% RSLogix 500 project 4P4_E_drbitboy_refactor_00.RSS, saved by version 8.30.00.16 %
PROJECT "4P4_E"    % processor: Bul.1763 MicroLogix 1100 Series B %

PROGRAM FILES
  LAD 2 "MAIN_PROG"  7 rungs
  LAD 3 "USER_FAULT"  2 rungs
  LAD 5 "INPUTCHECK"  10 rungs
  LAD 7 "DOBUSINESS"  13 rungs
  LAD 14 "OUTPUT2SIM"  3 rungs
  LAD 15 "SIMULATION"  20 rungs

DATA FILES
  O0 OUTPUT  4 elements
  I1 INPUT  6 elements
  S2 STATUS  66 elements
  B3 BINARY  32 elements
  T4 TIMER  40 elements
  C5 COUNTER  32 elements
  R6 CONTROL  16 elements
  N7 INTEGER  105 elements
  F8 FLOAT  1 elements

LADDER 2 "MAIN_PROG"
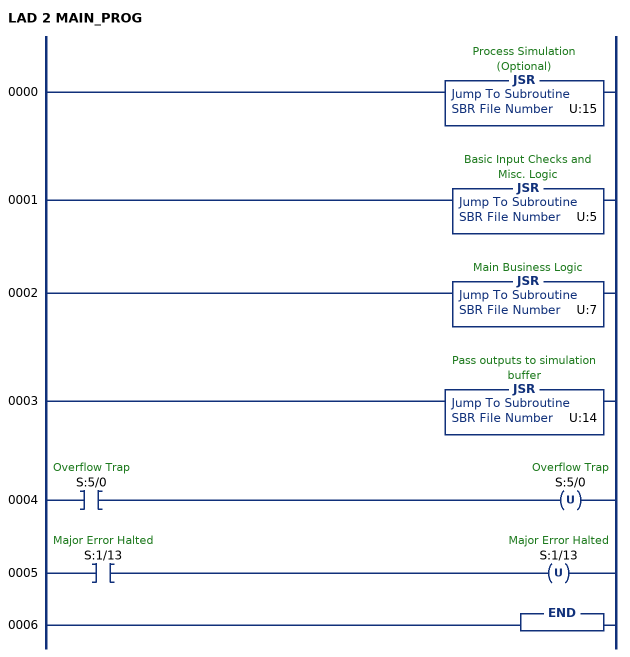
% Rung: 0 %
SOR JSR U:15 EOR
%   U:15  "Process Simulation (Optional)" %
% Rung: 1 %
SOR JSR U:5 EOR
%   U:5  "Basic Input Checks and Misc. Logic" %
% Rung: 2 %
SOR JSR U:7 EOR
%   U:7  "Main Business Logic" %
% Rung: 3 %
SOR JSR U:14 EOR
%   U:14  "Pass outputs to simulation buffer" %
% Rung: 4 %
SOR XIC S:5/0 OTU S:5/0 EOR
%   S:5/0  "Overflow Trap" %
% Rung: 5 %
SOR XIC S:1/13 OTU S:1/13 EOR
%   S:1/13  "Major Error Halted" %
% Rung: 6 %
SOR END EOR

LADDER 3 "USER_FAULT"
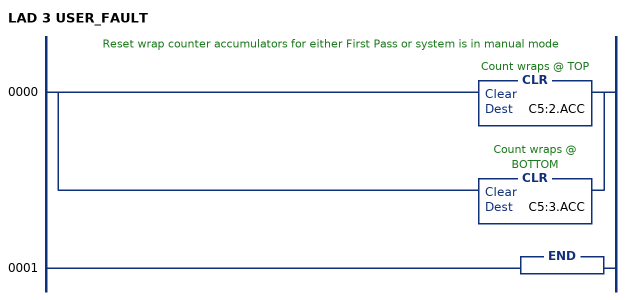
% Rung: 0 %
% Reset wrap counter accumulators for either First Pass or system is in manual mode %
SOR BST CLR C5:2.ACC NXB CLR C5:3.ACC BND EOR
%   C5:2  "Count wraps @ TOP" %
%   C5:3  "Count wraps @ BOTTOM" %
% Rung: 1 %
SOR END EOR

LADDER 5 "INPUTCHECK"
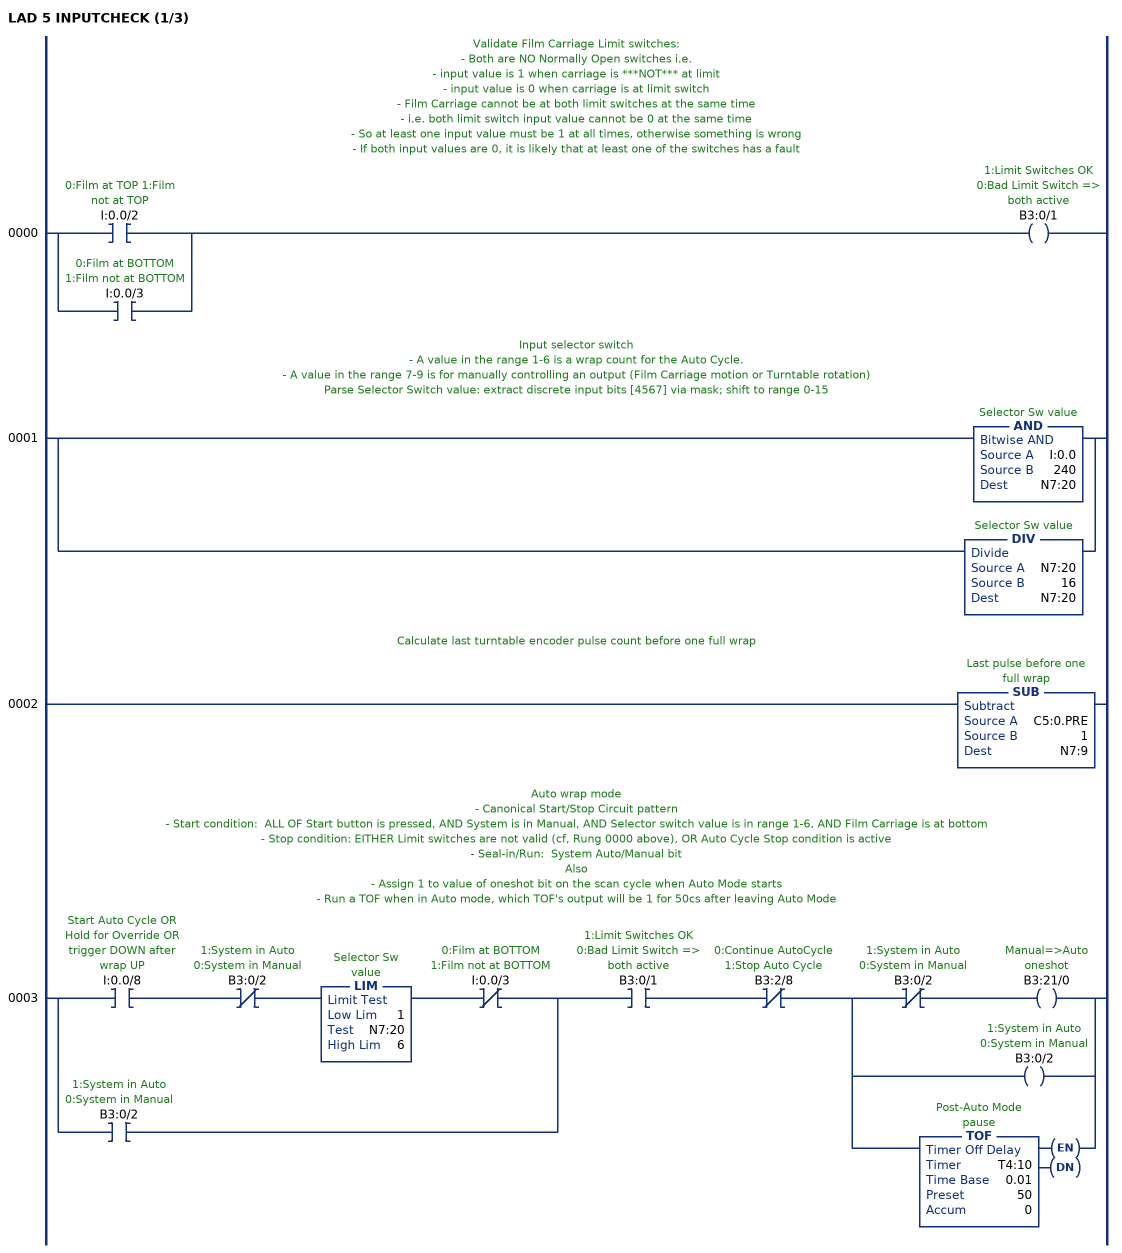
% Rung: 0 %
% Validate Film Carriage Limit switches:
% - Both are NO Normally Open switches i.e.
%   - input value is 1 when carriage is ***NOT*** at limit
%   - input value is 0 when carriage is at limit switch
% - Film Carriage cannot be at both limit switches at the same time
%   - i.e. both limit switch input value cannot be 0 at the same time
%   - So at least one input value must be 1 at all times, otherwise something is wrong
% - If both input values are 0, it is likely that at least one of the switches has a fault %
SOR BST XIC I:0.0/2 NXB XIC I:0.0/3 BND OTE B3:0/1 EOR
%   I:0.0/2  "0:Film at TOP 1:Film not at TOP" %
%   XIC I:0.0/2  "1:Film not at TOP" %
%   I:0.0/3  "0:Film at BOTTOM 1:Film not at BOTTOM" %
%   XIC I:0.0/3  "1:Film not at BOTTOM" %
%   B3:0/1  "1:Limit Switches OK 0:Bad Limit Switch => both active" %
% Rung: 1 %
% Input selector switch
% - A value in the range 1-6 is a wrap count for the Auto Cycle.
% - A value in the range 7-9 is for manually controlling an output (Film Carriage motion or Turntable rotation)
% 
% Parse Selector Switch value: extract discrete input bits [4567] via mask; shift to range 0-15 %
SOR BST AND I:0.0 240 N7:20 NXB DIV N7:20 16 N7:20 BND EOR
%   I:0.0  "INPUT Word" %
%   N7:20  "Selector Sw value" %
% Rung: 2 %
% Calculate last turntable encoder pulse count before one full wrap %
SOR SUB C5:0.PRE 1 N7:9 EOR
%   C5:0  "Count turntable pulses 112 per wrap?" %
%   N7:9  "Last pulse before one full wrap" %
% Rung: 3 %
% Auto wrap mode
% - Canonical Start/Stop Circuit pattern
%   - Start condition:  ALL OF Start button is pressed, AND System is in Manual, AND Selector switch value is in range 1-6, AND Film Carriage is at bottom
%   - Stop condition: EITHER Limit switches are not valid (cf, Rung 0000 above), OR Auto Cycle Stop condition is active
%   - Seal-in/Run:  System Auto/Manual bit
% Also
% - Assign 1 to value of oneshot bit on the scan cycle when Auto Mode starts
% - Run a TOF when in Auto mode, which TOF's output will be 1 for 50cs after leaving Auto Mode %
SOR BST XIC I:0.0/8 XIO B3:0/2 LIM 1 N7:20 6 XIO I:0.0/3 NXB XIC B3:0/2 BND XIC B3:0/1 XIO B3:2/8 BST XIO B3:0/2 OTE B3:21/0 NXB OTE B3:0/2 NXB TOF T4:10 0.01 50 0 BND EOR
%   I:0.0/8  "Start Auto Cycle OR Hold for Override OR trigger DOWN after wrap UP" %
%   B3:0/2  "1:System in Auto 0:System in Manual" %
%   XIO B3:0/2  "0:System in Manual" %
%   N7:20  "Selector Sw value" %
%   I:0.0/3  "0:Film at BOTTOM 1:Film not at BOTTOM" %
%   XIO I:0.0/3  "0:Film at BOTTOM" %
%   XIC B3:0/2  "1:System in Auto" %
%   B3:0/1  "1:Limit Switches OK 0:Bad Limit Switch => both active" %
%   XIC B3:0/1  "1:Limit Switches OK" %
%   B3:2/8  "0:Continue AutoCycle 1:Stop Auto Cycle" %
%   B3:21/0  "Manual=>Auto oneshot" %
%   T4:10  "Post-Auto Mode pause" %

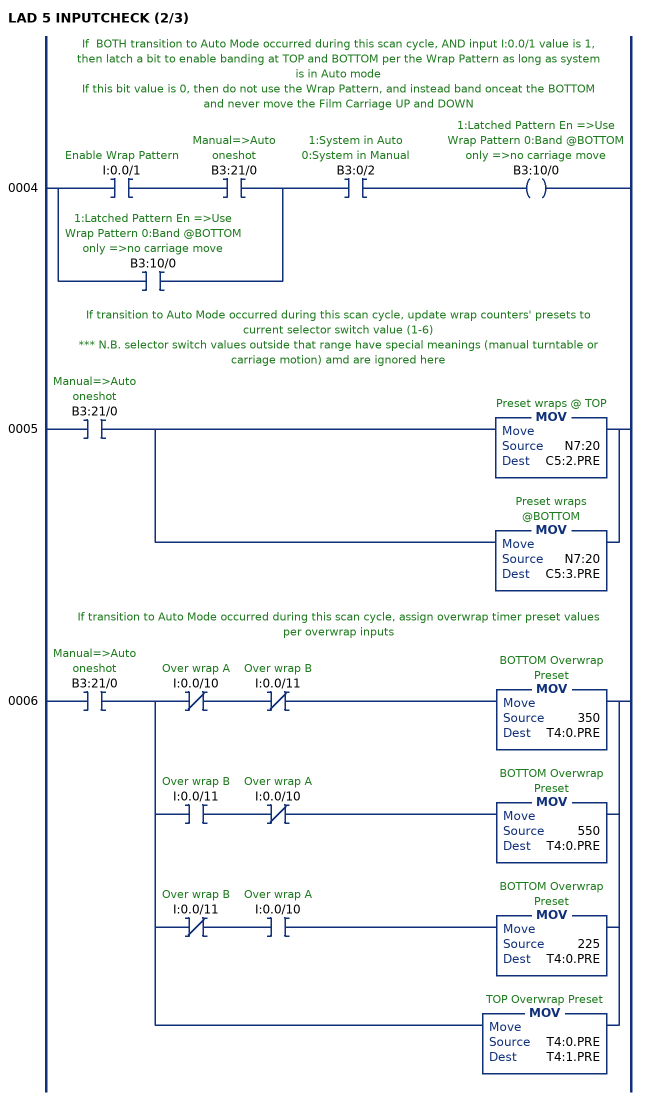
% Rung: 4 %
% If  BOTH transition to Auto Mode occurred during this scan cycle, AND input I:0.0/1 value is 1, then latch a bit to enable banding at TOP and BOTTOM per the Wrap Pattern as long as system is in Auto mode
% If this bit value is 0, then do not use the Wrap Pattern, and instead band onceat the BOTTOM and never move the Film Carriage UP and DOWN %
SOR BST XIC I:0.0/1 XIC B3:21/0 NXB XIC B3:10/0 BND XIC B3:0/2 OTE B3:10/0 EOR
%   I:0.0/1  "Enable Wrap Pattern" %
%   B3:21/0  "Manual=>Auto oneshot" %
%   B3:10/0  "1:Latched Pattern En =>Use Wrap Pattern 0:Band @BOTTOM only =>no carriage move" %
%   XIC B3:10/0  "1:Latched Pattern En =>Use Wrap Pattern =>In Auto Mode" %
%   B3:0/2  "1:System in Auto 0:System in Manual" %
%   XIC B3:0/2  "1:System in Auto" %
% Rung: 5 %
% If transition to Auto Mode occurred during this scan cycle, update wrap counters' presets to current selector switch value (1-6)
% *** N.B. selector switch values outside that range have special meanings (manual turntable or carriage motion) amd are ignored here %
SOR XIC B3:21/0 BST MOV N7:20 C5:2.PRE NXB MOV N7:20 C5:3.PRE BND EOR
%   B3:21/0  "Manual=>Auto oneshot" %
%   N7:20  "Selector Sw value" %
%   C5:2.PRE  "Preset wraps @ TOP" %
%   C5:3.PRE  "Preset wraps @BOTTOM" %
% Rung: 6 %
% If transition to Auto Mode occurred during this scan cycle, assign overwrap timer preset values per overwrap inputs %
SOR XIC B3:21/0 BST XIO I:0.0/10 XIO I:0.0/11 MOV 350 T4:0.PRE NXB XIC I:0.0/11 XIO I:0.0/10 MOV 550 T4:0.PRE NXB XIO I:0.0/11 XIC I:0.0/10 MOV 225 T4:0.PRE NXB MOV T4:0.PRE T4:1.PRE BND EOR
%   B3:21/0  "Manual=>Auto oneshot" %
%   I:0.0/10  "Over wrap A" %
%   I:0.0/11  "Over wrap B" %
%   T4:0.PRE  "BOTTOM Overwrap Preset" %
%   T4:1.PRE  "TOP Overwrap Preset" %

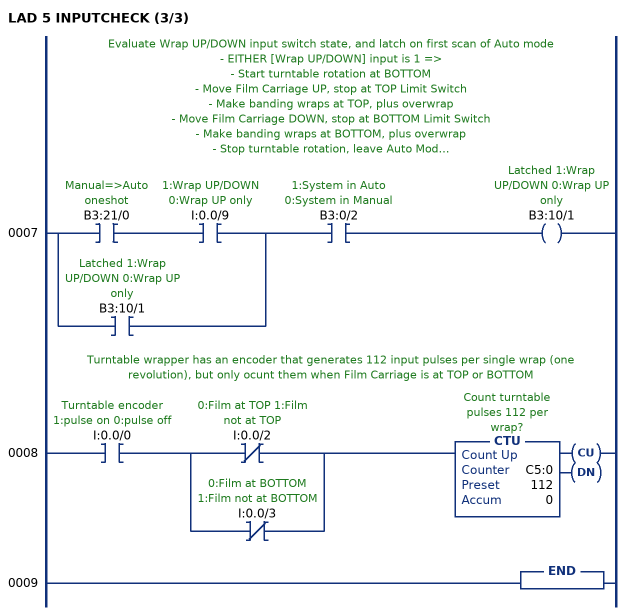
% Rung: 7 %
% Evaluate Wrap UP/DOWN input switch state, and latch on first scan of Auto mode
% - EITHER [Wrap UP/DOWN] input is 1 =>
%   - Start turntable rotation at BOTTOM
%   - Move Film Carriage UP, stop at TOP Limit Switch
%   - Make banding wraps at TOP, plus overwrap
%   - Move Film Carriage DOWN, stop at BOTTOM Limit Switch
%   - Make banding wraps at BOTTOM, plus overwrap
%   - Stop turntable rotation, leave Auto Mode
% - OR [Wrap UP/DOWN] input is 0 (Wrap UP only) =>
%   - Start turntable rotation at BOTTOM
%   - Make banding wraps at BOTTOM, plus overwrap
%   - Move File Carriage UP, stop at TOP Limit Switch
%   - Make banding wraps at TOP, plus overwrap
%   - Stop Turntable rotation
%   - Flash light, wait for operator to (cut film and then) press Start
%   - Move Film Carriage DOWN, stop at BOTTOM Limit Switch
%   - Leave Auto Mode %
SOR BST XIC B3:21/0 XIC I:0.0/9 NXB XIC B3:10/1 BND XIC B3:0/2 OTE B3:10/1 EOR
%   B3:21/0  "Manual=>Auto oneshot" %
%   I:0.0/9  "1:Wrap UP/DOWN 0:Wrap UP only" %
%   B3:10/1  "Latched 1:Wrap UP/DOWN 0:Wrap UP only" %
%   XIC B3:10/1  "Latched 1:Wrap UP/DOWN" %
%   B3:0/2  "1:System in Auto 0:System in Manual" %
%   XIC B3:0/2  "1:System in Auto" %
% Rung: 8 %
% Turntable wrapper has an encoder that generates 112 input pulses per single wrap (one revolution), but only ocunt them when Film Carriage is at TOP or BOTTOM %
SOR XIC I:0.0/0 BST XIO I:0.0/2 NXB XIO I:0.0/3 BND CTU C5:0 112 0 EOR
%   I:0.0/0  "Turntable encoder 1:pulse on 0:pulse off" %
%   XIC I:0.0/0  "1:Turntable encoder pulse on" %
%   I:0.0/2  "0:Film at TOP 1:Film not at TOP" %
%   XIO I:0.0/2  "0:Film at TOP" %
%   I:0.0/3  "0:Film at BOTTOM 1:Film not at BOTTOM" %
%   XIO I:0.0/3  "0:Film at BOTTOM" %
%   C5:0  "Count turntable pulses 112 per wrap?" %
% Rung: 9 %
SOR END EOR

LADDER 7 "DOBUSINESS"
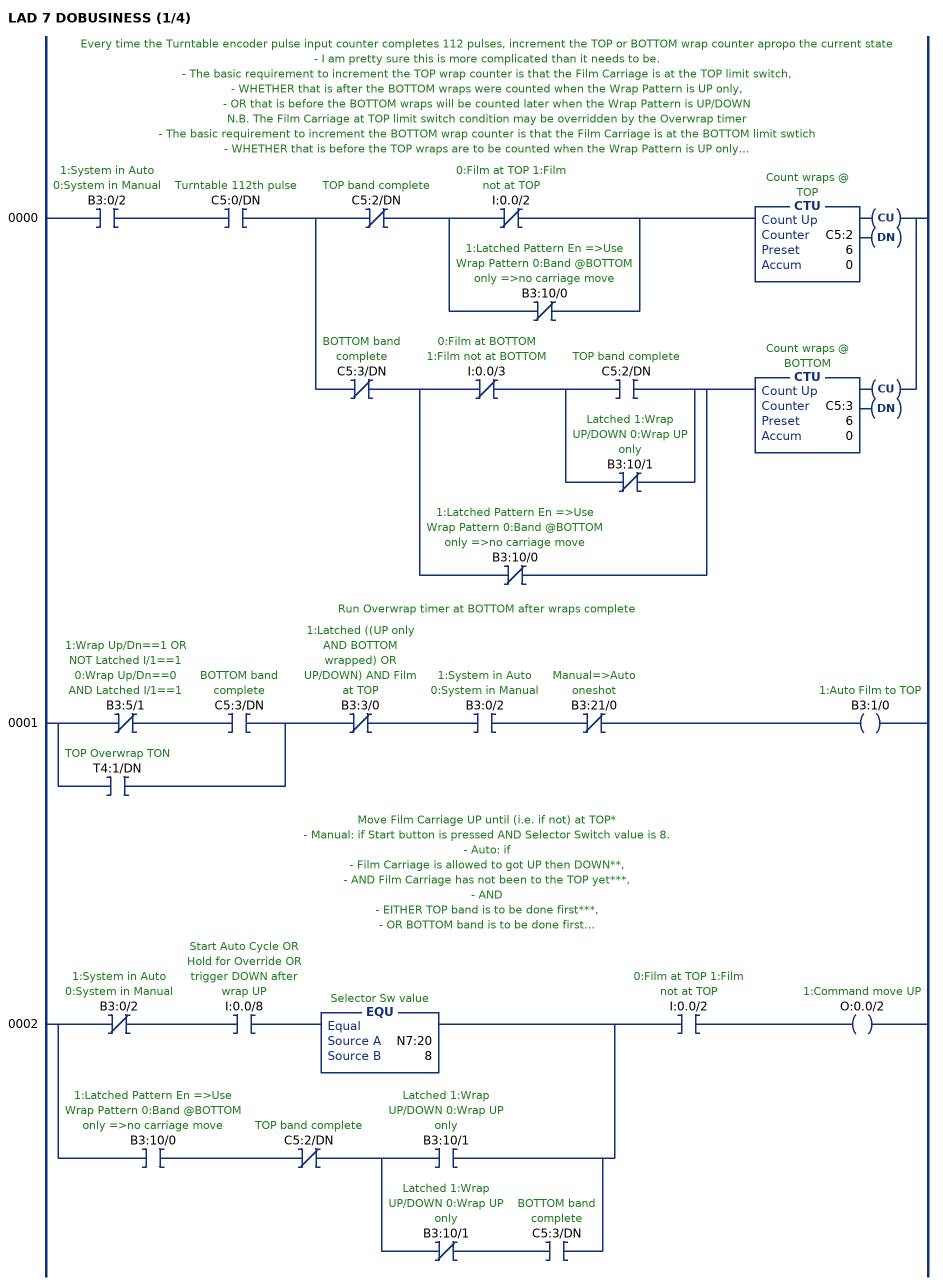
% Rung: 0 %
% Every time the Turntable encoder pulse input counter completes 112 pulses, increment the TOP or BOTTOM wrap counter apropo the current state
% - I am pretty sure this is more complicated than it needs to be.
% 
% - The basic requirement to increment the TOP wrap counter is that the Film Carriage is at the TOP limit switch,
%   - WHETHER that is after the BOTTOM wraps were counted when the Wrap Pattern is UP only,
%   - OR that is before the BOTTOM wraps will be counted later when the Wrap Pattern is UP/DOWN
% N.B. The Film Carriage at TOP limit switch condition may be overridden by the Overwrap timer
% 
% - The basic requirement to increment the BOTTOM wrap counter is that the Film Carriage is at the BOTTOM limit swtich
%   - WHETHER that is before the TOP wraps are to be counted when the Wrap Pattern is UP only,
%   - OR that is after the TOP wraps were counted when the Wrap Pattern is UP/DOWN
% N.B. the TOP wraps completed check for Wrap Pattern UP/DOWN may be overriden by the T4:6 timer done bit when inpu I:0.0/1 value is 0 %
SOR XIC B3:0/2 XIC C5:0/DN BST XIO C5:2/DN BST XIO I:0.0/2 NXB XIO B3:10/0 BND CTU C5:2 6 0 NXB XIO C5:3/DN BST XIO I:0.0/3 BST XIC C5:2/DN NXB XIO B3:10/1 BND NXB XIO B3:10/0 BND CTU C5:3 6 0 BND EOR
%   B3:0/2  "1:System in Auto 0:System in Manual" %
%   XIC B3:0/2  "1:System in Auto" %
%   C5:0/DN  "Turntable 112th pulse" %
%   C5:2/DN  "TOP band complete" %
%   XIO C5:2/DN  "TOP band incomplete" %
%   I:0.0/2  "0:Film at TOP 1:Film not at TOP" %
%   XIO I:0.0/2  "0:Film at TOP" %
%   B3:10/0  "1:Latched Pattern En =>Use Wrap Pattern 0:Band @BOTTOM only =>no carriage move" %
%   XIO B3:10/0  "0:Band @BOTTOM only =>no carriage move" %
%   C5:2  "Count wraps @ TOP" %
%   C5:3/DN  "BOTTOM band complete" %
%   XIO C5:3/DN  "BOTTOM band incomplete" %
%   I:0.0/3  "0:Film at BOTTOM 1:Film not at BOTTOM" %
%   XIO I:0.0/3  "0:Film at BOTTOM" %
%   B3:10/1  "Latched 1:Wrap UP/DOWN 0:Wrap UP only" %
%   XIO B3:10/1  "Latched 0:Wrap UP only" %
%   C5:3  "Count wraps @ BOTTOM" %
% Rung: 1 %
% Run Overwrap timer at BOTTOM after wraps complete %
SOR BST XIO B3:5/1 XIC C5:3/DN NXB XIC T4:1/DN BND XIO B3:3/0 XIC B3:0/2 XIO B3:21/0 OTE B3:1/0 EOR
%   B3:5/1  "1:Wrap Up/Dn==1 OR NOT Latched I/1==1 0:Wrap Up/Dn==0 AND Latched I/1==1" %
%   XIO B3:5/1  "0:Wrap UP only AND Latched I/1==1" %
%   C5:3/DN  "BOTTOM band complete" %
%   T4:1  "TOP Overwrap TON" %
%   B3:3/0  "1:Latched ((UP only AND BOTTOM wrapped) OR UP/DOWN) AND Film at TOP" %
%   B3:0/2  "1:System in Auto 0:System in Manual" %
%   XIC B3:0/2  "1:System in Auto" %
%   B3:21/0  "Manual=>Auto oneshot" %
%   XIO B3:21/0  "0:Start btn released in Auto mode" %
%   B3:1/0  "1:Auto Film to TOP" %
% Rung: 2 %
% Move Film Carriage UP until (i.e. if not) at TOP*
% - Manual: if Start button is pressed AND Selector Switch value is 8.
% - Auto: if
%   - Film Carriage is allowed to got UP then DOWN**,
%   - AND Film Carriage has not been to the TOP yet***,
%   - AND
%     - EITHER TOP band is to be done first***,
%     - OR BOTTOM band is to be done first.
% 
% * Don't need to check if Limit Switches are OK because [Film not at TOP] ensures they are
% ** [Latched Wrap Pattern Enabled] is only 1 if already in Auto Mode
% *** [TOP band incomplete] will be 1when to stop Film Carriage moving up when it is at BOTTOM the second time for [Wrap UP/DOWN]. %
SOR BST XIO B3:0/2 XIC I:0.0/8 EQU N7:20 8 NXB XIC B3:10/0 XIO C5:2/DN BST XIC B3:10/1 NXB XIO B3:10/1 XIC C5:3/DN BND BND XIC I:0.0/2 OTE O:0.0/2 EOR
%   B3:0/2  "1:System in Auto 0:System in Manual" %
%   XIO B3:0/2  "0:System in Manual" %
%   I:0.0/8  "Start Auto Cycle OR Hold for Override OR trigger DOWN after wrap UP" %
%   N7:20  "Selector Sw value" %
%   B3:10/0  "1:Latched Pattern En =>Use Wrap Pattern 0:Band @BOTTOM only =>no carriage move" %
%   XIC B3:10/0  "1:Latched Pattern En =>Use Wrap Pattern =>In Auto Mode" %
%   C5:2/DN  "TOP band complete" %
%   XIO C5:2/DN  "TOP band incomplete" %
%   B3:10/1  "Latched 1:Wrap UP/DOWN 0:Wrap UP only" %
%   XIC B3:10/1  "Latched 1:Wrap UP/DOWN" %
%   XIO B3:10/1  "Latched 0:Wrap UP only" %
%   C5:3/DN  "BOTTOM band complete" %
%   I:0.0/2  "0:Film at TOP 1:Film not at TOP" %
%   XIC I:0.0/2  "1:Film not at TOP" %
%   O:0.0/2  "1:Command move UP" %

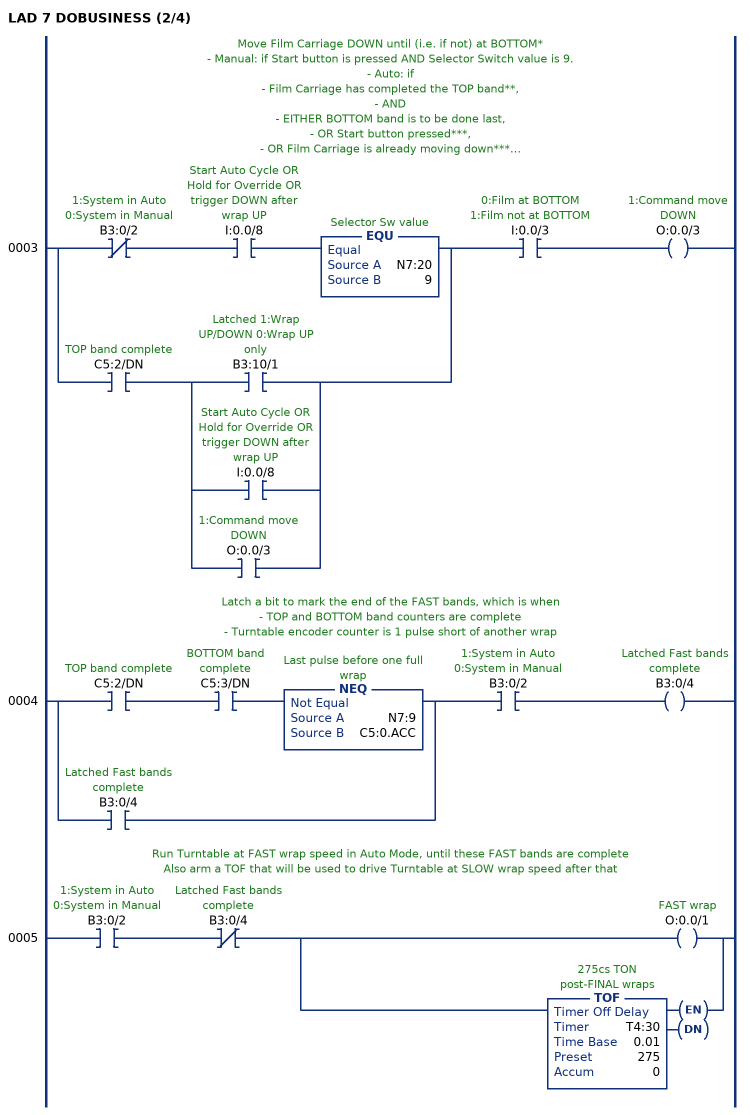
% Rung: 3 %
% Move Film Carriage DOWN until (i.e. if not) at BOTTOM*
% - Manual: if Start button is pressed AND Selector Switch value is 9.
% - Auto: if
%   - Film Carriage has completed the TOP band**,
%   - AND
%     - EITHER BOTTOM band is to be done last,
%     - OR Start button pressed***,
%     - OR Film Carriage is already moving down***.
% 
% * Don't need to check if Limit Switches are OK because [Film not at BOTTOM] ensures they are
% ** Film Carriage would not be away from BOTTOM unless [Wrap Pattern Enabled]
%   - Also TOP band can only be complete if system is in Auto Mode, because TOP band count is cleared to 0 in Manual
% *** Those last two will be the case when Wrap Pattern is Wrap UP only %
SOR BST XIO B3:0/2 XIC I:0.0/8 EQU N7:20 9 NXB XIC C5:2/DN BST XIC B3:10/1 NXB XIC I:0.0/8 NXB XIC O:0.0/3 BND BND XIC I:0.0/3 OTE O:0.0/3 EOR
%   B3:0/2  "1:System in Auto 0:System in Manual" %
%   XIO B3:0/2  "0:System in Manual" %
%   I:0.0/8  "Start Auto Cycle OR Hold for Override OR trigger DOWN after wrap UP" %
%   N7:20  "Selector Sw value" %
%   C5:2/DN  "TOP band complete" %
%   B3:10/1  "Latched 1:Wrap UP/DOWN 0:Wrap UP only" %
%   XIC B3:10/1  "Latched 1:Wrap UP/DOWN" %
%   O:0.0/3  "1:Command move DOWN" %
%   I:0.0/3  "0:Film at BOTTOM 1:Film not at BOTTOM" %
%   XIC I:0.0/3  "1:Film not at BOTTOM" %
% Rung: 4 %
% Latch a bit to mark the end of the FAST bands, which is when
% - TOP and BOTTOM band counters are complete
% - Turntable encoder counter is 1 pulse short of another wrap %
SOR BST XIC C5:2/DN XIC C5:3/DN NEQ N7:9 C5:0.ACC NXB XIC B3:0/4 BND XIC B3:0/2 OTE B3:0/4 EOR
%   C5:2/DN  "TOP band complete" %
%   C5:3/DN  "BOTTOM band complete" %
%   N7:9  "Last pulse before one full wrap" %
%   C5:0.ACC  "Turntable pulse count" %
%   B3:0/4  "Latched Fast bands complete" %
%   XIC B3:0/4  "1:Fast bands complete" %
%   B3:0/2  "1:System in Auto 0:System in Manual" %
%   XIC B3:0/2  "1:System in Auto" %
% Rung: 5 %
% Run Turntable at FAST wrap speed in Auto Mode, until these FAST bands are complete
% Also arm a TOF that will be used to drive Turntable at SLOW wrap speed after that %
SOR XIC B3:0/2 XIO B3:0/4 BST OTE O:0.0/1 NXB TOF T4:30 0.01 275 0 BND EOR
%   B3:0/2  "1:System in Auto 0:System in Manual" %
%   XIC B3:0/2  "1:System in Auto" %
%   B3:0/4  "Latched Fast bands complete" %
%   XIO B3:0/4  "0:Fast bands incomplete" %
%   O:0.0/1  "FAST wrap" %
%   T4:30  "275cs TON post-FINAL wraps" %

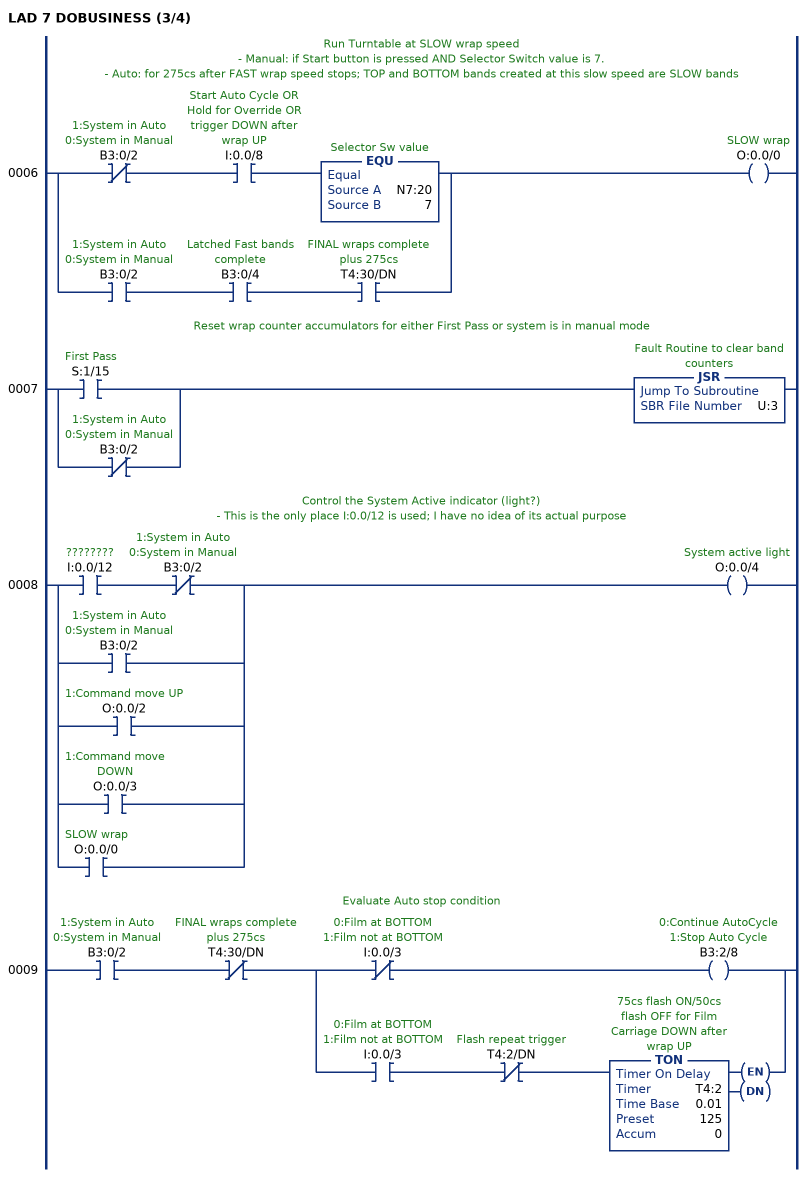
% Rung: 6 %
% Run Turntable at SLOW wrap speed
% - Manual: if Start button is pressed AND Selector Switch value is 7.
% - Auto: for 275cs after FAST wrap speed stops; TOP and BOTTOM bands created at this slow speed are SLOW bands %
SOR BST XIO B3:0/2 XIC I:0.0/8 EQU N7:20 7 NXB XIC B3:0/2 XIC B3:0/4 XIC T4:30/DN BND OTE O:0.0/0 EOR
%   B3:0/2  "1:System in Auto 0:System in Manual" %
%   XIO B3:0/2  "0:System in Manual" %
%   I:0.0/8  "Start Auto Cycle OR Hold for Override OR trigger DOWN after wrap UP" %
%   N7:20  "Selector Sw value" %
%   XIC B3:0/2  "1:System in Auto" %
%   B3:0/4  "Latched Fast bands complete" %
%   XIC B3:0/4  "1:Fast bands complete" %
%   T4:30/DN  "FINAL wraps complete plus 275cs" %
%   O:0.0/0  "SLOW wrap" %
% Rung: 7 %
% Reset wrap counter accumulators for either First Pass or system is in manual mode %
SOR BST XIC S:1/15 NXB XIO B3:0/2 BND JSR U:3 EOR
%   S:1/15  "First Pass" %
%   B3:0/2  "1:System in Auto 0:System in Manual" %
%   XIO B3:0/2  "0:System in Manual" %
%   U:3  "Fault Routine to clear band counters" %
% Rung: 8 %
% Control the System Active indicator (light?)
% - This is the only place I:0.0/12 is used; I have no idea of its actual purpose %
SOR BST XIC I:0.0/12 XIO B3:0/2 NXB XIC B3:0/2 NXB XIC O:0.0/2 NXB XIC O:0.0/3 NXB XIC O:0.0/0 BND OTE O:0.0/4 EOR
%   I:0.0/12  "????????" %
%   B3:0/2  "1:System in Auto 0:System in Manual" %
%   XIO B3:0/2  "0:System in Manual" %
%   XIC B3:0/2  "1:System in Auto" %
%   O:0.0/2  "1:Command move UP" %
%   O:0.0/3  "1:Command move DOWN" %
%   O:0.0/0  "SLOW wrap" %
%   O:0.0/4  "System active light" %
% Rung: 9 %
% Evaluate Auto stop condition %
SOR XIC B3:0/2 XIO T4:30/DN BST XIO I:0.0/3 OTE B3:2/8 NXB XIC I:0.0/3 XIO T4:2/DN TON T4:2 0.01 125 0 BND EOR
%   B3:0/2  "1:System in Auto 0:System in Manual" %
%   XIC B3:0/2  "1:System in Auto" %
%   T4:30/DN  "FINAL wraps complete plus 275cs" %
%   I:0.0/3  "0:Film at BOTTOM 1:Film not at BOTTOM" %
%   XIO I:0.0/3  "0:Film at BOTTOM" %
%   B3:2/8  "0:Continue AutoCycle 1:Stop Auto Cycle" %
%   XIC I:0.0/3  "1:Film not at BOTTOM" %
%   T4:2/DN  "Flash repeat trigger" %
%   T4:2  "75cs flash ON/50cs flash OFF for Film Carriage DOWN after wrap UP" %

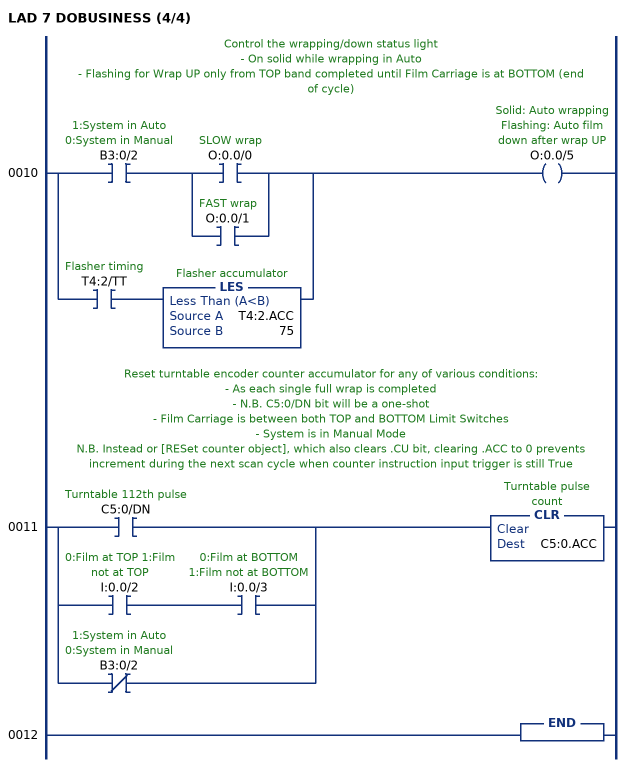
% Rung: 10 %
% Control the wrapping/down status light
% - On solid while wrapping in Auto
% - Flashing for Wrap UP only from TOP band completed until Film Carriage is at BOTTOM (end of cycle) %
SOR BST XIC B3:0/2 BST XIC O:0.0/0 NXB XIC O:0.0/1 BND NXB XIC T4:2/TT LES T4:2.ACC 75 BND OTE O:0.0/5 EOR
%   B3:0/2  "1:System in Auto 0:System in Manual" %
%   XIC B3:0/2  "1:System in Auto" %
%   O:0.0/0  "SLOW wrap" %
%   O:0.0/1  "FAST wrap" %
%   T4:2/TT  "Flasher timing" %
%   T4:2.ACC  "Flasher accumulator" %
%   O:0.0/5  "Solid: Auto wrapping Flashing: Auto film down after wrap UP" %
% Rung: 11 %
% Reset turntable encoder counter accumulator for any of various conditions:
% - As each single full wrap is completed
%   - N.B. C5:0/DN bit will be a one-shot
% - Film Carriage is between both TOP and BOTTOM Limit Switches
% - System is in Manual Mode
% N.B. Instead or [RESet counter object], which also clears .CU bit, clearing .ACC to 0 prevents
%          increment during the next scan cycle when counter instruction input trigger is still True %
SOR BST XIC C5:0/DN NXB XIC I:0.0/2 XIC I:0.0/3 NXB XIO B3:0/2 BND CLR C5:0.ACC EOR
%   C5:0/DN  "Turntable 112th pulse" %
%   I:0.0/2  "0:Film at TOP 1:Film not at TOP" %
%   XIC I:0.0/2  "1:Film not at TOP" %
%   I:0.0/3  "0:Film at BOTTOM 1:Film not at BOTTOM" %
%   XIC I:0.0/3  "1:Film not at BOTTOM" %
%   B3:0/2  "1:System in Auto 0:System in Manual" %
%   XIO B3:0/2  "0:System in Manual" %
%   C5:0.ACC  "Turntable pulse count" %
% Rung: 12 %
SOR END EOR

LADDER 14 "OUTPUT2SIM"
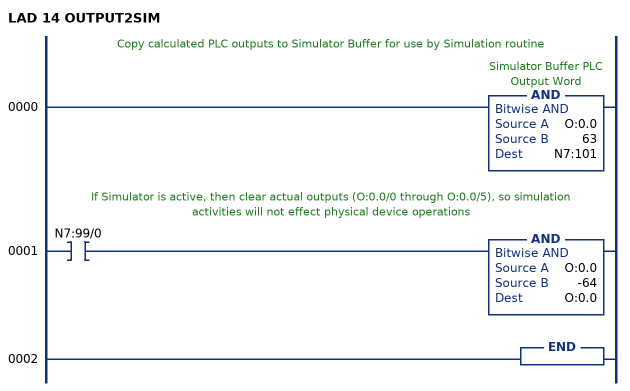
% Rung: 0 %
% Copy calculated PLC outputs to Simulator Buffer for use by Simulation routine %
SOR AND O:0.0 63 N7:101 EOR
%   N7:101  "Simulator Buffer PLC Output Word" %
% Rung: 1 %
% If Simulator is active, then clear actual outputs (O:0.0/0 through O:0.0/5), so simulation activities will not effect physical device operations %
SOR XIC N7:99/0 AND O:0.0 -64 O:0.0 EOR
% Rung: 2 %
SOR END EOR

LADDER 15 "SIMULATION"
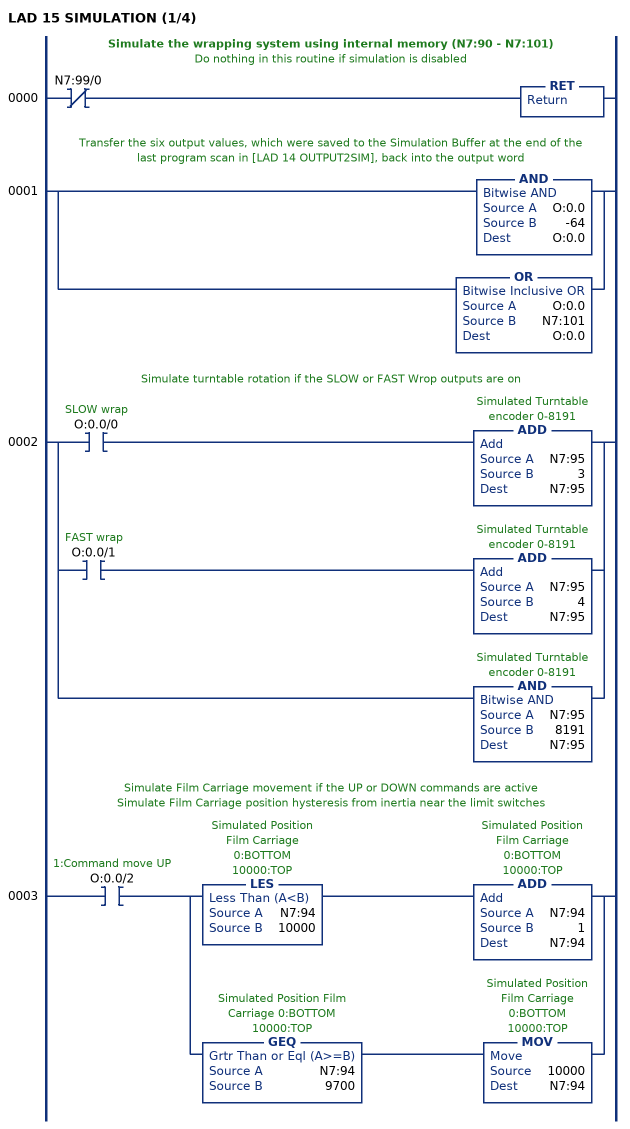
% Rung: 0 %
% TITLE: Simulate the wrapping system using internal memory (N7:90 - N7:101) %
% Do nothing in this routine if simulation is disabled %
SOR XIO N7:99/0 RET EOR
% Rung: 1 %
% Transfer the six output values, which were saved to the Simulation Buffer at the end of the last program scan in [LAD 14 OUTPUT2SIM], back into the output word %
SOR BST AND O:0.0 -64 O:0.0 NXB OR O:0.0 N7:101 O:0.0 BND EOR
%   N7:101  "Simulator Buffer PLC Output Word" %
% Rung: 2 %
% Simulate turntable rotation if the SLOW or FAST Wrop outputs are on %
SOR BST XIC O:0.0/0 ADD N7:95 3 N7:95 NXB XIC O:0.0/1 ADD N7:95 4 N7:95 NXB AND N7:95 8191 N7:95 BND EOR
%   O:0.0/0  "SLOW wrap" %
%   N7:95  "Simulated Turntable encoder 0-8191" %
%   O:0.0/1  "FAST wrap" %
% Rung: 3 %
% Simulate Film Carriage movement if the UP or DOWN commands are active
% Simulate Film Carriage position hysteresis from inertia near the limit switches %
SOR XIC O:0.0/2 BST LES N7:94 10000 ADD N7:94 1 N7:94 NXB GEQ N7:94 9700 MOV 10000 N7:94 BND EOR
%   O:0.0/2  "1:Command move UP" %
%   N7:94  "Simulated Position Film Carriage 0:BOTTOM 10000:TOP" %

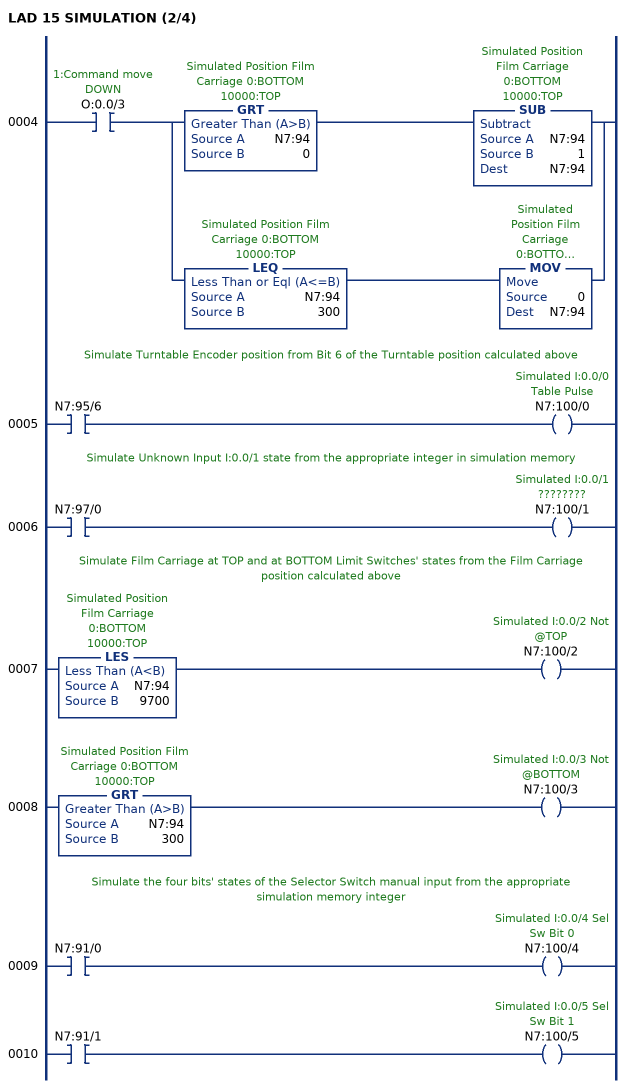
% Rung: 4 %
SOR XIC O:0.0/3 BST GRT N7:94 0 SUB N7:94 1 N7:94 NXB LEQ N7:94 300 MOV 0 N7:94 BND EOR
%   O:0.0/3  "1:Command move DOWN" %
%   N7:94  "Simulated Position Film Carriage 0:BOTTOM 10000:TOP" %
% Rung: 5 %
% Simulate Turntable Encoder position from Bit 6 of the Turntable position calculated above %
SOR XIC N7:95/6 OTE N7:100/0 EOR
%   N7:100/0  "Simulated I:0.0/0 Table Pulse" %
% Rung: 6 %
% Simulate Unknown Input I:0.0/1 state from the appropriate integer in simulation memory %
SOR XIC N7:97/0 OTE N7:100/1 EOR
%   N7:100/1  "Simulated I:0.0/1 ????????" %
% Rung: 7 %
% Simulate Film Carriage at TOP and at BOTTOM Limit Switches' states from the Film Carriage position calculated above %
SOR LES N7:94 9700 OTE N7:100/2 EOR
%   N7:94  "Simulated Position Film Carriage 0:BOTTOM 10000:TOP" %
%   N7:100/2  "Simulated I:0.0/2 Not @TOP" %
% Rung: 8 %
SOR GRT N7:94 300 OTE N7:100/3 EOR
%   N7:94  "Simulated Position Film Carriage 0:BOTTOM 10000:TOP" %
%   N7:100/3  "Simulated I:0.0/3 Not @BOTTOM" %
% Rung: 9 %
% Simulate the four bits' states of the Selector Switch manual input from the appropriate simulation memory integer %
SOR XIC N7:91/0 OTE N7:100/4 EOR
%   N7:100/4  "Simulated I:0.0/4 Sel Sw Bit 0" %
% Rung: 10 %
SOR XIC N7:91/1 OTE N7:100/5 EOR
%   N7:100/5  "Simulated I:0.0/5 Sel Sw Bit 1" %

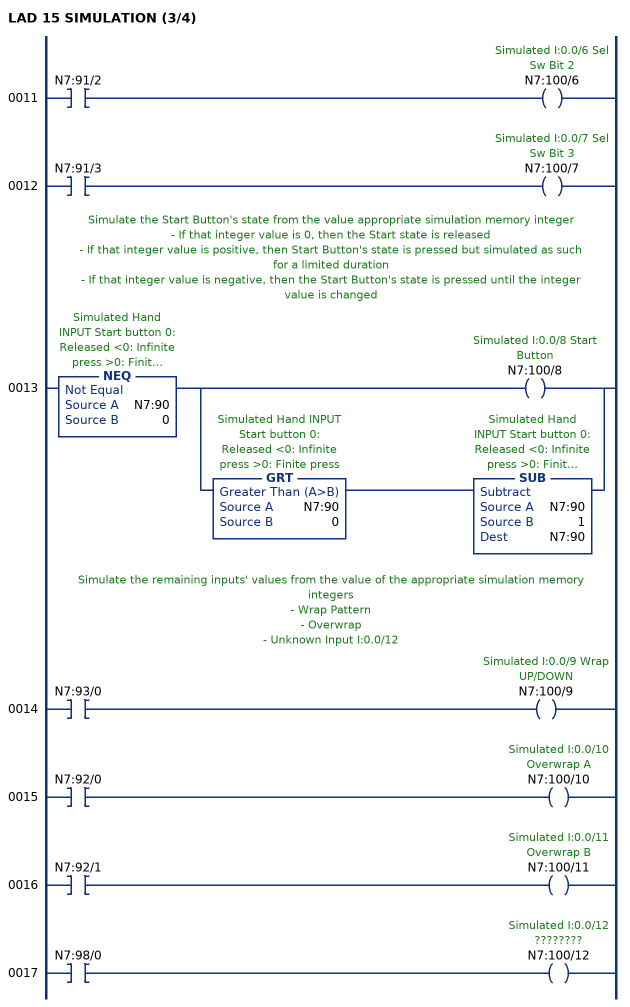
% Rung: 11 %
SOR XIC N7:91/2 OTE N7:100/6 EOR
%   N7:100/6  "Simulated I:0.0/6 Sel Sw Bit 2" %
% Rung: 12 %
SOR XIC N7:91/3 OTE N7:100/7 EOR
%   N7:100/7  "Simulated I:0.0/7 Sel Sw Bit 3" %
% Rung: 13 %
% Simulate the Start Button's state from the value appropriate simulation memory integer
% - If that integer value is 0, then the Start state is released
% - If that integer value is positive, then Start Button's state is pressed but simulated as such for a limited duration
% - If that integer value is negative, then the Start Button's state is pressed until the integer value is changed %
SOR NEQ N7:90 0 BST OTE N7:100/8 NXB GRT N7:90 0 SUB N7:90 1 N7:90 BND EOR
%   N7:90  "Simulated Hand INPUT Start button 0: Released <0: Infinite press >0: Finite press" %
%   N7:100/8  "Simulated I:0.0/8 Start Button" %
% Rung: 14 %
% Simulate the remaining inputs' values from the value of the appropriate simulation memory integers
% - Wrap Pattern
% - Overwrap
% - Unknown Input I:0.0/12 %
SOR XIC N7:93/0 OTE N7:100/9 EOR
%   N7:100/9  "Simulated I:0.0/9 Wrap UP/DOWN" %
% Rung: 15 %
SOR XIC N7:92/0 OTE N7:100/10 EOR
%   N7:100/10  "Simulated I:0.0/10 Overwrap A" %
% Rung: 16 %
SOR XIC N7:92/1 OTE N7:100/11 EOR
%   N7:100/11  "Simulated I:0.0/11 Overwrap B" %
% Rung: 17 %
SOR XIC N7:98/0 OTE N7:100/12 EOR
%   N7:100/12  "Simulated I:0.0/12 ????????" %

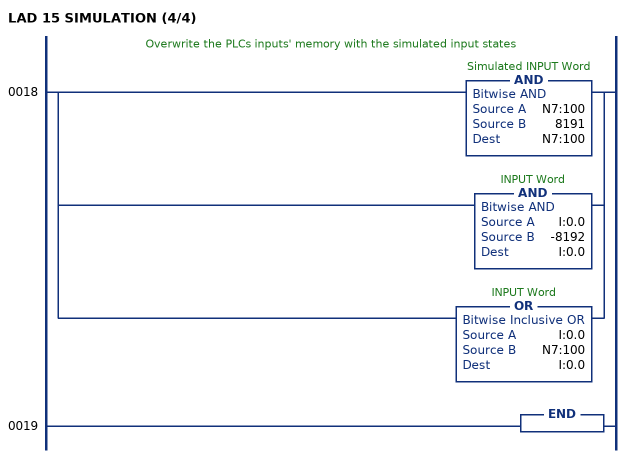
% Rung: 18 %
% Overwrite the PLCs inputs' memory with the simulated input states %
SOR BST AND N7:100 8191 N7:100 NXB AND I:0.0 -8192 I:0.0 NXB OR I:0.0 N7:100 I:0.0 BND EOR
%   N7:100  "Simulated INPUT Word" %
%   I:0.0  "INPUT Word" %
% Rung: 19 %
SOR END EOR

OTHER DOCUMENTED ADDRESSES
  B3:0/0  "1:Trigger pulse count reset"
  B3:0/3  "1:Latched FINAL wraps done + 375cs + 111 pulses 0:Continue wrapping"
  B3:0/12  "2:Latch move film DOWN after wrap UP"
  B3:1/1  "1:Wraps incomplete AND System in Auto +50cs 0:Wraps complete OR Sys in Manual"
  B3:1/8  "Film carriage DOWN trigger"
  B3:2/6  "1:Latched FINAL wraps done plus 275cs AND wrapping 0:Wraps incomplete OR NOT wrapping"
  B3:3/1  "1:Latched TOP wrapped AND film at BOTTOM"
  B3:4/0  "First-pass one-shot"
  B3:5/0  "1:Start button triggers Auto; Count switch=1-6 0:Start button other Count switch=7-9"
  B3:8/2  "Raise Film Carriage (UP override) 1: Count switch at 8 and Start pressed"
  B3:8/3  "Lower Film Carriage (DOWN override) 1: Count switch at 9 and Start pressed"
  B3:8/9  "Rotate turntable (Wrap override) 1:Count switch at 7 and Start pressed"
  B3:9/0  "FINAL wraps complete"
  I:0.0/4  "Count bit 0 Value=1"
  I:0.0/5  "Count bit 1 Value=2"
  I:0.0/6  "Count bit 2 Value = 4"
  I:0.0/7  "Count bit 3 Value=8"
  N7:36  "BOTTOM wraps remaining"
  N7:37  "TOP wraps remaining"
  N7:91  "Simulated Hand INPUT Selector switch 1-6:Wrap count 7:Rotate 8:UP 9:DOWN"
  N7:92  "Simulated Hand INPUT Overwrap 0:Off 1:Low 2:High"
  N7:93  "Simulated Hand INPUT Wrap pattern 0:UP  1:UP/DOWN"
  N7:96  "Simulate Film Carriage Inertia and Limit Switch Hysteresis"
  N7:97  "Simulated INPUT I:0.0/1 ???????? Bit 0"
  N7:98  "Simulated INPUT I:0.0/12 ???????? Bit 0"
  N7:99  "0:Disable Simulation 1:Use Simulation"
  N7:101/0  "Simulator Buffer SLOW wrap?"
  N7:101/1  "Simulator Buffer FAST wrap?"
  N7:101/2  "Simulator Buffer 1:Command move UP"
  N7:101/3  "Simulator Buffer 1:Command move DOWN"
  N7:101/4  "Simulator Buffer System active light"
  N7:101/5  "Simulator Buffer Solid: Auto wrapping Flashing: Auto film down after wrap UP"
  T4:0  "BOTTOM Overwrap TON"
  T4:0/DN  "Overwrap after I/1=0 @50cs latch"
  T4:3  "50cs flash ON film DOWN after wrap UP"
  T4:4  "50cs TON of Auto AND wraps incomplete"
  T4:6  "10cs TON NOT Latched I/1==1 in Auto"
  T4:6/DN  "10cs NOT Latched I/1==1"
  T4:7  "10+10cs TON NOT Latched I/1==1 in Auto"
  T4:7/DN  "20cs NOT Latched I/1==1"
  T4:8  "50cs Latched TON in Auto mode with I/1=0"
  T4:8/DN  "50cs Latched I/1==0"

OTHER INSTRUCTION COMMENTS
  B3:5/0 XIC  "1:Start button triggers Auto; Count switch=1-6"
  B3:2/8 XIC  "1:Stop Auto Cycle"
  B3:0/3 XIO  "0:Continue wrapping"
  B3:0/3 XIC  "1:Latched wraps done"
  N7:37 LES  "No more TOP wraps"
  N7:36 LES  "No more BOTTOM wraps"
  B3:5/1 XIC  "1:Wrap UP/DOWN OR NOT Latched I/1==1"
  T4:3/DN XIO  "75cs flash OFF film DOWN after wrap UP"
  B3:1/1 XIC  "1:Wraps incomplete AND System in Auto +50cs"
  B3:2/6 XIO  "0:Wraps incomplete OR NOT wrapping"
  B3:2/6 XIC  "1:Latched (FINAL wraps done +275cs) AND wrapping"
  I:0.0/0 XIO  "0:Turntable encoder pulse off"

DATA TABLE (non-zero values as saved)
DATA T4
% .PRE .ACC %
% T4:0 % 350 0
% T4:1 % 10 0
% T4:2 % 125 0
% T4:3 % 50 0
% T4:4 % 50 0
% T4:6 % 10 0
% T4:7 % 10 0
% T4:8 % 50 0
% T4:9 % 100 0
% T4:10 % 50 0
% T4:11 % 275 0
% T4:12 % 20 0
% T4:13 % 400 400
% T4:14 % 400 0
% T4:15 % 150 150
% T4:16 % 300 300
% T4:17 % 120 0
% T4:18 % 150 0
% T4:19 % 200 0
% T4:20 % 100 0
% T4:21 % 50 0
% T4:22 % 100 0
% T4:23 % 70 0
% T4:24 % 10 0
% T4:25 % 100 0
% T4:26 % 300 0
% T4:27 % 100 0
% T4:29 % 1 1
% T4:30 % 275 0
% T4:31 % 450 0
% T4:32 % 50 50
% T4:34 % 200 0
% T4:36 % 800 0
% T4:37 % 200 0
% T4:38 % 350 0
DATA C5
% .PRE .ACC %
% C5:0 % 112 0
% C5:1 % 9999 1456
% C5:2 % 6 0
% C5:3 % 6 0
% C5:4 % 9999 221
% C5:5 % 9999 0
% C5:6 % 1 0
% C5:7 % 9999 7
% C5:8 % 3 0
% C5:9 % 3 0
% C5:10 % 20 1
% C5:11 % 9999 0
% C5:12 % 9999 2
% C5:14 % 76 0
% C5:15 % 3 0
% C5:16 % 2 1
DATA R6
% .LEN .POS %
% R6:0 % 16 0
DATA N7
% N7:0 % 2 2 2 0 0 0 1 221 112 111
% N7:10 % 80 1 0 0 0 0 0 0 0 0
% N7:90 % 0 2 0 0 0 0 0 1 0 0
